Staubli VAL3: readArea.pgx

public program readArea(num x_nIdArea, num x_nDBnumber, num x_nStartAt, num x_nQty, num& x_nBuffer[])
  local num l_Address
  local num l_nElementsNum
  local num l_nIndex
  local num l_nLength
  local num l_nMaxElements
  local num l_nOffs
  local num l_nS7R[31]
  local num l_nSizeReq
  local num l_nTempDec
  local num l_nToIndex
  local num l_nTotElements
  local num l_nWordSize
  local string l_sRes
  local string l_sTempBin
begin

  //Header begin

  //This function read a memory area from the PLC starting from "x_nStartAt" byte and for a "x_nQty" number of bytes.
  //The result is stored in a "num" array where each element is a byte of the memory area read.
  //
  //Input parameters
  //
  //num x_nIdArea: the PLC's memory area identifier (you'll find several identifier as public members of the library with the suffix "nArea").
	//num x_nDBnumber: the DB number you're reading from (this parameter is not important if you're not reading a db...but in VAL3 there's no possibility to overload functions so we must pass it the same to this function!).
	//num x_nStartAt:: the byte adddress you want start to read from.
	//num x_nQty: the amount of bytes you want to read.
  //
  //Output parameters
  // num x_nBuffer[1]:  a monodimensional array where the area read is stored. If the size of this buffer is smaller than "x_nQty" only "size(x_nBuffer[])" will be read .
  //
  //Examples
  //
  // call S7:readArea(S7:nAreaDB,nDBread,2,1,l_nRes)
  //
  //History
  // Creation: 24-12-16 - Alessio Villa
  //Header end

  l_nOffs=0
  l_nWordSize=1

  call setLastError(nNoErrors)

  if size(x_nBuffer)<x_nQty
    //small buffer
    x_nQty=size(x_nBuffer)
  endIf

  if x_nIdArea==nAreaCT or x_nIdArea==nAreaTM
    l_nWordSize=2
  endIf

  //18 is the reply header size
  l_nMaxElements=(nPDULength-18)/l_nWordSize
  l_nTotElements=x_nQty

  while l_nTotElements>0 and nLastError==nNoErrors

    l_nElementsNum=l_nTotElements
    if l_nElementsNum>l_nMaxElements
      l_nElementsNum=l_nMaxElements
    endIf
    //calc request size
    l_nSizeReq=l_nElementsNum*l_nWordSize

    //setup the telegram!
    getData("nS7_R",l_nS7R)

    //set area number
    l_nS7R[27]=x_nIdArea
    if x_nIdArea==nAreaDB
      //set db number
      l_sTempBin=""
      call bitOp:DecToBin(x_nDBnumber,l_sTempBin)
      call bitOp:shiftRight(l_sTempBin,8)
      l_nTempDec=0
      call bitOp:BinToDec(l_sTempBin,l_nTempDec)
      l_nS7R[25]=l_nTempDec
      l_sTempBin=""
      call bitOp:DecToBin(x_nDBnumber,l_sTempBin)
      l_sRes=""
      call bitOp:boolAnd(l_sTempBin,"0000000011111111",l_sRes)
      l_nTempDec=0
      call bitOp:BinToDec(l_sRes,l_nTempDec)
      l_nS7R[26]=l_nTempDec
    endIf

    // Adjusts Start and word length
    if x_nIdArea==nAreaCT or x_nIdArea==nAreaTM
      l_Address=x_nStartAt
      if x_nIdArea==nAreaCT
        l_nS7R[22]=nWLcounter
      else
        l_nS7R[22]=nWLtimer
      endIf
    else
      //shift left 3 bit
      l_Address=x_nStartAt*power(2,3)
    endIf

    //number of elements
    l_nS7R[23]=l_nElementsNum*power(2,8)
    l_nS7R[24]=l_nElementsNum
    //address in plc
    l_sTempBin=""
    call bitOp:DecToBin(l_Address,l_sTempBin)
    l_sRes=""
    call bitOp:boolAnd(l_sTempBin,"0000000011111111",l_sRes)
    l_nTempDec=0
    call bitOp:BinToDec(l_sRes,l_nTempDec)
    l_nS7R[30]=l_nTempDec
    call bitOp:shiftRight(l_sTempBin,8)

    l_sRes=""
    call bitOp:boolAnd(l_sTempBin,"0000000011111111",l_sRes)
    l_nTempDec=0
    call bitOp:BinToDec(l_sRes,l_nTempDec)
    l_nS7R[29]=l_nTempDec
    call bitOp:shiftRight(l_sTempBin,8)

    l_sRes=""
    call bitOp:boolAnd(l_sTempBin,"0000000011111111",l_sRes)
    l_nTempDec=0
    call bitOp:BinToDec(l_sRes,l_nTempDec)
    l_nS7R[28]=l_nTempDec

    //send the telegram!
    call sendPacket(l_nS7R,nRDsize)
    if nLastError==nNoErrors
      call recvISOpacket(l_nLength)
      if nLastError==nNoErrors
        if l_nLength>=18
          //if ((Length-18==SizeRequested) && (PDU.H[31]==0xFF))
          if l_nLength-18==l_nSizeReq and PDU.S7telegram.H[14]==255
            //copy data in the target buffer
            l_nIndex=0
            if size(x_nBuffer)-l_nOffs<size(PDU.S7telegram.DATA)
              l_nToIndex=size(x_nBuffer)-l_nOffs-1
            else
              l_nToIndex=size(PDU.S7telegram.DATA)-1
            endIf
            for l_nIndex=0 to l_nToIndex
              x_nBuffer[l_nOffs+l_nIndex]=PDU.S7telegram.DATA[l_nIndex]
            endFor
            l_nOffs=l_nOffs+l_nSizeReq
          else
            call setLastError(nErrDataRead)
          endIf
        else
          call setLastError(nErrISOInvPDU)
        endIf
      else
        //error detected
      endIf
    else
      call setLastError(nErrTCPSend)
    endIf

    l_nTotElements=l_nTotElements-l_nElementsNum
    x_nStartAt=x_nStartAt+l_nElementsNum*l_nWordSize

  endWhile

end
